(* CoDeSys 2.3 export: TP_FB.EXP *)

(* POU TP_FB, ST *)
FUNCTION_BLOCK TP_FB
VAR_INPUT
	on_intlk : BOOL;
	on_ena : BOOL;
	off_ena : BOOL;

	on_req : BOOL;
	off_req : BOOL;
END_VAR
VAR_OUTPUT
	on_cmd : BOOL;
	not_symbol : BOOL;
END_VAR
VAR
END_VAR
on_cmd 		:=	on_intlk AND
				(NOT (off_ena AND off_req)) AND
				((on_ena AND on_req) OR on_cmd);

not_symbol	:=	(on_cmd AND NOT off_ena) OR
				(NOT on_cmd AND NOT (on_intlk AND on_ena));
END_FUNCTION_BLOCK
